// TIA Portal V16 export
// export: Created 2021-09-08T12:44:32.7351686Z, ExportSetting WithDefaults, DisplayName Totally Integrated Automation Portal, DisplayVersion V16 Update 3, DisplayName TIA Portal Version Control Interface, DisplayVersion V16 Update 2, DisplayName TIA Portal Openness, DisplayVersion V16 Update 3, DisplayName TIA Portal Teamcenter Gateway, DisplayVersion V16, DisplayName STEP 7 Professional, DisplayVersion V16 Update 3, DisplayName STEP 7 Safety, DisplayVersion V16, DisplayName WinCC Advanced, DisplayVersion V16 Update 3
VAR_GLOBAL   // PLC tag table "A10_AQ"
   aqDP101 AT %QW68 : Int;   // DP101 Завдання
   aqDP502 AT %QW70 : Int;   // DP502 Завдання
   aqDP501 AT %QW72 : Int;   // DP501 Завдання
   aqDP801 AT %QW74 : Int;   // DP801 Завдання
   aqDP802 AT %QW76 : Int;   // DP802 Завдання
   aqDP803 AT %QW78 : Int;   // DP803 Завдання
   aqDP1001 AT %QW80 : Int;   // DP1001 Завдання
   PQW18_Reserve AT %QW82 : Int;   // Резерв
END_VAR
VAR_GLOBAL CONSTANT   // user constants
   "qwDP-101" : Int := 0;
   "qwDP-502" : Int := 1;
   "qwDP-501" : Int := 2;
   "qwDP-801" : Int := 3;
   "qwDP-802" : Int := 4;
   "qwDP-803" : Int := 5;
   "qwDP-1001" : Int := 6;
   qw18_Reserve : Int := 7;
END_VAR
